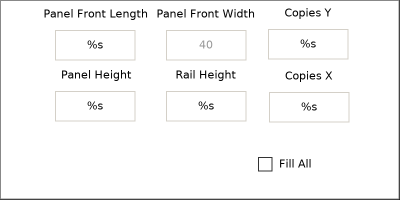
VISUALIZATION V_ProductionArona  // 400x200
VAR_IN_OUT
	HMI : ST_PackMLBaseModule_HMI;
	HMI_GantryXYZ : ST_GantryXYZ_HMI;
	HMI_Recipe : ST_RecipeBuilder_HMI;
END_VAR
    RoundedRectangle (0,0 400x200)
    Textfield (55,30 80x30), "%s", text variable: HMI_Recipe.Config.PanelFrontLength
        OnMouseClick: write the text variable via VisuDialogs.Numpad, min HMI_Recipe.Limits.PanelFrontLength.MinVal, max HMI_Recipe.Limits.PanelFrontLength.MaxVal
    Label (38,4 116x20), "Panel Front Length"
    Textfield (166,30 80x30), "40"
        OnMouseClick: write the text variable via VisuDialogs.Numpad, min HMI_Recipe.Limits.PanelFrontWidth.MinVal, max HMI_Recipe.Limits.PanelFrontWidth.MaxVal
    Label (117,4 178x20), "Panel Front Width"
    Textfield (55,91 80x30), "%s", text variable: HMI_Recipe.Config.PanelHeight
        OnMouseClick: write the text variable via VisuDialogs.Numpad, min HMI_Recipe.Limits.PanelHeight.MinVal, max HMI_Recipe.Limits.PanelHeight.MaxVal
    Label (39,65 115x20), "Panel Height"
    Textfield (166,91 80x30), "%s", text variable: HMI_Recipe.Config.RailHeightCorrection
        OnMouseClick: write the text variable via VisuDialogs.Numpad, min HMI_Recipe.Limits.RailHeightCorrection.MinVal, max HMI_Recipe.Limits.RailHeightCorrection.MaxVal
    Label (155,65 102x20), "Rail Height"
    Checkbox (256,149 72x30), "Fill All", variable: HMI_Recipe.Config.FillAll
    Textfield (269,92 80x30), "%s", text variable: HMI_Recipe.Config.RequestedCopiesX, input disabled if: MAIN.Seedra.RecipeConfig_HMI.Config.FillAll
        OnMouseClick: write the text variable via VisuDialogs.Numpad, min 1, max MAIN.Seedra.RecipeConfig_HMI.Limits.RequestedCopiesX.MaxVal
    Label (258,66 102x20), "Copies X"
    Textfield (268,29 80x30), "%s", text variable: HMI_Recipe.Config.RequestedCopiesY, input disabled if: MAIN.Seedra.RecipeConfig_HMI.Config.FillAll
        OnMouseClick: write the text variable via VisuDialogs.Numpad, min 1, max MAIN.Seedra.RecipeConfig_HMI.Limits.RequestedCopiesY.MaxVal
    Label (257,3 102x20), "Copies Y"
END_VISUALIZATION

(* stored: Version 1.1.0.1, ProductVersion 3.1.4024.15
   Visu V_ProductionArona: Id {e190c579-abc8-43d7-84da-7a962e614c8d} *)
